(* Logix 5000 project; controller EuniceF_ICA16 vendor 1 type 14 code 150 rev 37.11; software revision 37.00 *)

TASK MainTask (continuous, watchdog 500 ms) : MainProgram

MODULES
   Local : vendor 1 type 14 code 150 (Compact 0, rev 37.11)
      Discrete_IO : Embedded (Compact 1, rev 3.1, Output RPI 20 ms)
      Analog_IO : Embedded (Compact 2, rev 1.1, Output RPI 80 ms)
      Counters : Embedded (Compact 3, rev 1.1, Output RPI 20 ms)
END_MODULES

VAR_GLOBAL   (* controller tags *)
   Motor : ALIAS FOR Local:1:O.Data.1;
   seq : DINT;
   START : ALIAS FOR Local:1:I.Data.11;
   STEP : ALIAS FOR Local:1:I.Data.12;
   STOP : ALIAS FOR Local:1:I.Data.9;
END_VAR

PROGRAM MainProgram   (* main routine MainRoutine *)

ROUTINE MainRoutine   (* ladder *)
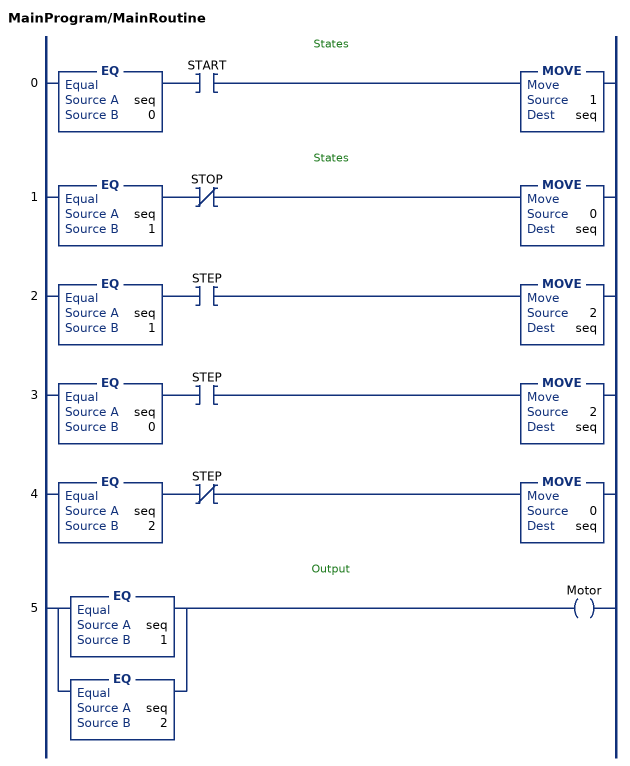
   // States
   0: EQ(seq,0)XIC(START)MOVE(1,seq);
   // States
   1: EQ(seq,1)XIO(STOP)MOVE(0,seq);
   2: EQ(seq,1)XIC(STEP)MOVE(2,seq);
   3: EQ(seq,0)XIC(STEP)MOVE(2,seq);
   4: EQ(seq,2)XIO(STEP)MOVE(0,seq);
   // Output
   5: [EQ(seq,1) ,EQ(seq,2) ]OTE(Motor);
END_ROUTINE
END_PROGRAM
